PROGRAM Fixt2_Seq_Call
VAR
	Clamp_1: FB_CylinderModule;
	Clamp_2: FB_CylinderModule;
	Clamp_3: FB_CylinderModule;
	Clamp_4: FB_CylinderModule;
	Clamp_5: FB_CylinderModule;
	Clamp_6: FB_CylinderModule;
	sAlwaysoff: BOOL;
	FB_AutoSeq_0: FB_AutoSeq;
	alwayson:BOOL;
	partmonitor:FB_PartMonitoring_fixt2;
	trunion:FB_Trunion;
END_VAR
VAR // added by the converter: edge detectors and wires of the graphical bodies
    _w1, _w2, _w3, _w4, _w5, _w6 : BOOL;
END_VAR

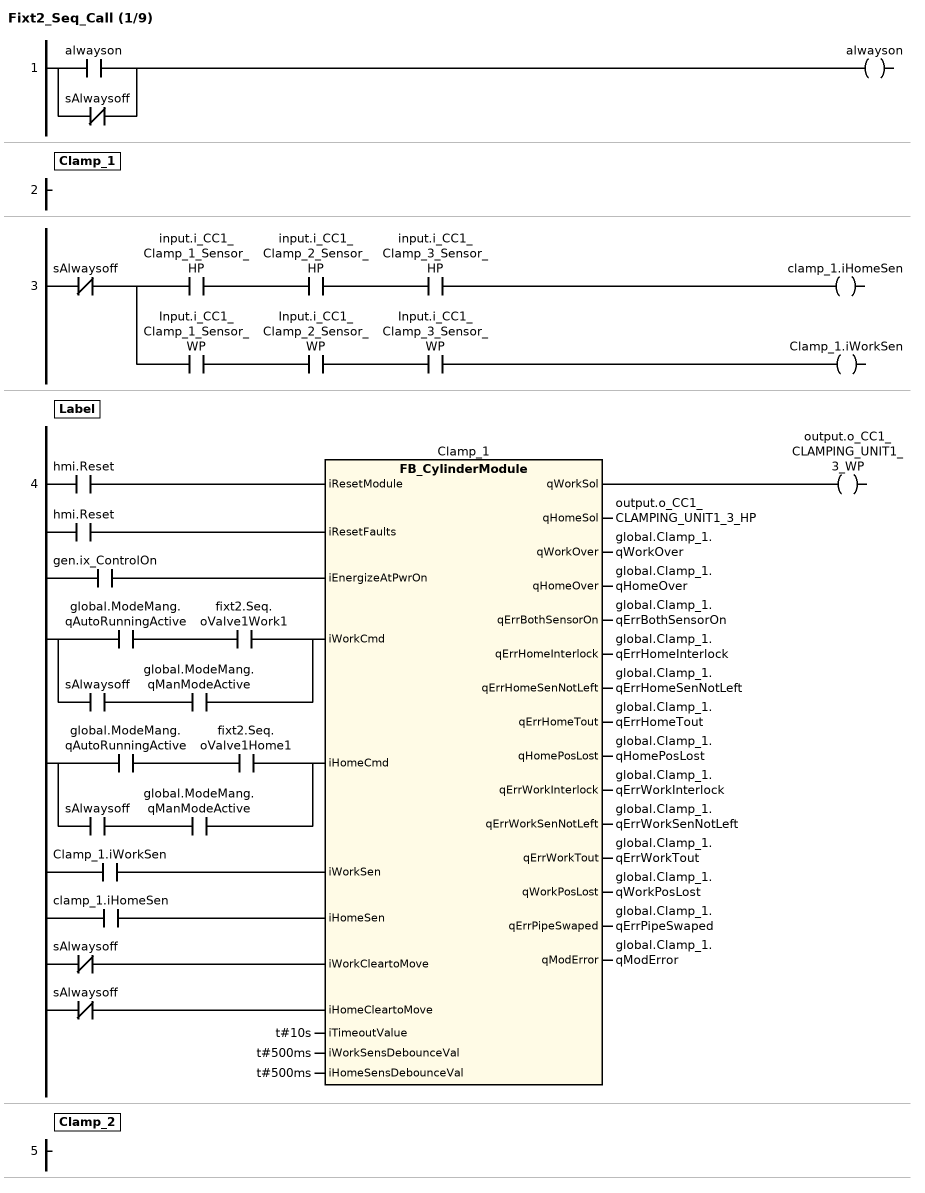
// NETWORK 1
alwayson := alwayson OR NOT sAlwaysoff;

// NETWORK 2
Clamp_1: ;

// NETWORK 3
_w1 := NOT sAlwaysoff;
clamp_1.iHomeSen := _w1 AND input.i_CC1_Clamp_1_Sensor_HP AND input.i_CC1_Clamp_2_Sensor_HP AND input.i_CC1_Clamp_3_Sensor_HP;
Clamp_1.iWorkSen := _w1 AND Input.i_CC1_Clamp_1_Sensor_WP AND Input.i_CC1_Clamp_2_Sensor_WP AND Input.i_CC1_Clamp_3_Sensor_WP;

// NETWORK 4
Label:
Clamp_1(
    iResetModule := hmi.Reset,
    iResetFaults := hmi.Reset,
    iEnergizeAtPwrOn := gen.ix_ControlOn,
    iWorkCmd := global.ModeMang.qAutoRunningActive AND fixt2.Seq.oValve1Work1 OR sAlwaysoff AND global.ModeMang.qManModeActive,
    iHomeCmd := global.ModeMang.qAutoRunningActive AND fixt2.Seq.oValve1Home1 OR sAlwaysoff AND global.ModeMang.qManModeActive,
    iWorkSen := Clamp_1.iWorkSen,
    iHomeSen := clamp_1.iHomeSen,
    iWorkCleartoMove := NOT sAlwaysoff,
    iHomeCleartoMove := NOT sAlwaysoff,
    iTimeoutValue := t#10s,
    iWorkSensDebounceVal := t#500ms,
    iHomeSensDebounceVal := t#500ms,
    qHomeSol => output.o_CC1_CLAMPING_UNIT1_3_HP,
    qWorkOver => global.Clamp_1.qWorkOver,
    qHomeOver => global.Clamp_1.qHomeOver,
    qErrBothSensorOn => global.Clamp_1.qErrBothSensorOn,
    qErrHomeInterlock => global.Clamp_1.qErrHomeInterlock,
    qErrHomeSenNotLeft => global.Clamp_1.qErrHomeSenNotLeft,
    qErrHomeTout => global.Clamp_1.qErrHomeTout,
    qHomePosLost => global.Clamp_1.qHomePosLost,
    qErrWorkInterlock => global.Clamp_1.qErrWorkInterlock,
    qErrWorkSenNotLeft => global.Clamp_1.qErrWorkSenNotLeft,
    qErrWorkTout => global.Clamp_1.qErrWorkTout,
    qWorkPosLost => global.Clamp_1.qWorkPosLost,
    qErrPipeSwaped => global.Clamp_1.qErrPipeSwaped,
    qModError => global.Clamp_1.qModError); // FB_CylinderModule
output.o_CC1_CLAMPING_UNIT1_3_WP := Clamp_1.qWorkSol;

// NETWORK 5
Clamp_2: ;

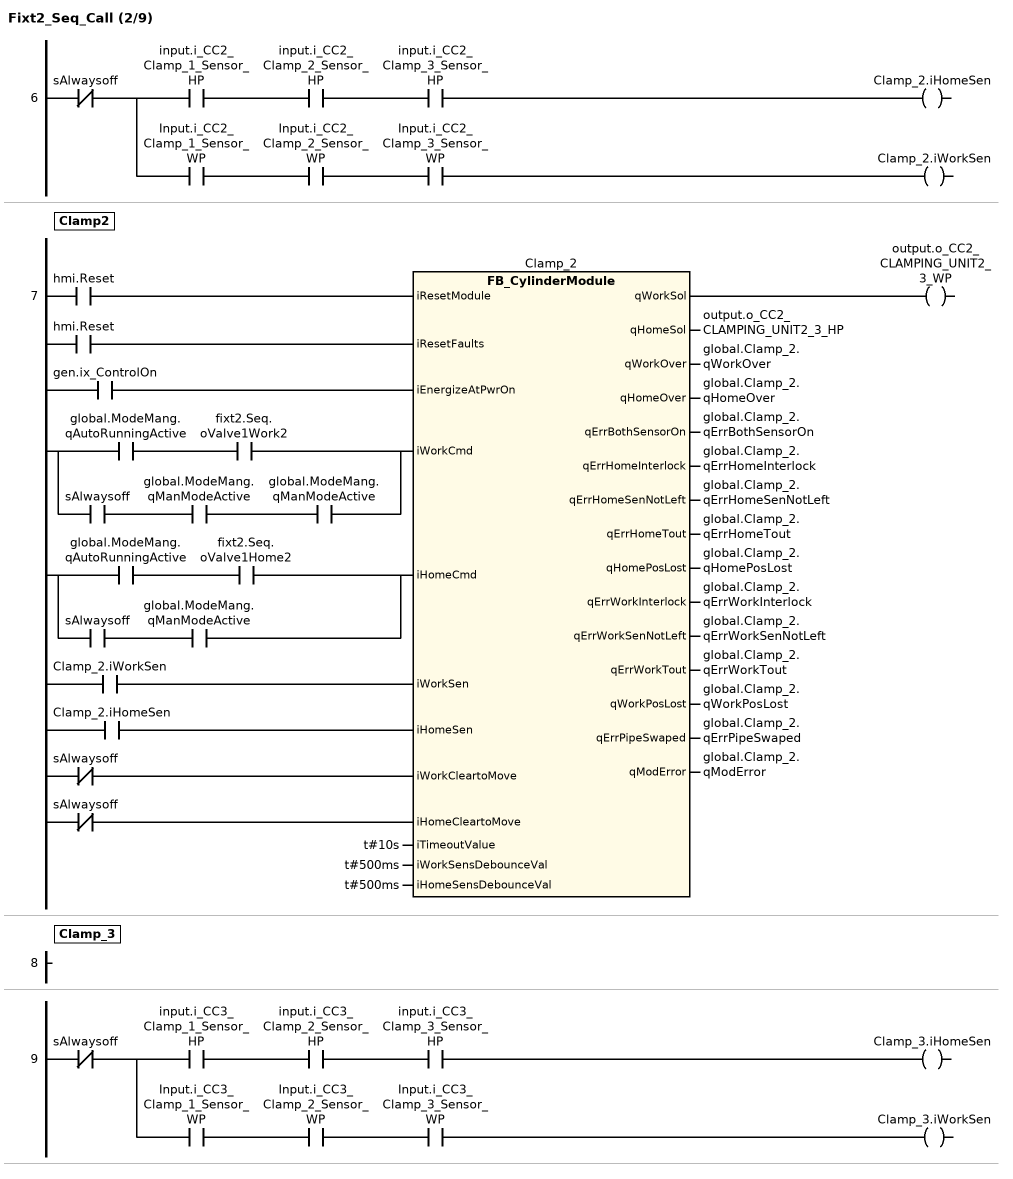
// NETWORK 6
_w2 := NOT sAlwaysoff;
Clamp_2.iHomeSen := _w2 AND input.i_CC2_Clamp_1_Sensor_HP AND input.i_CC2_Clamp_2_Sensor_HP AND input.i_CC2_Clamp_3_Sensor_HP;
Clamp_2.iWorkSen := _w2 AND Input.i_CC2_Clamp_1_Sensor_WP AND Input.i_CC2_Clamp_2_Sensor_WP AND Input.i_CC2_Clamp_3_Sensor_WP;

// NETWORK 7
Clamp2:
Clamp_2(
    iResetModule := hmi.Reset,
    iResetFaults := hmi.Reset,
    iEnergizeAtPwrOn := gen.ix_ControlOn,
    iWorkCmd := global.ModeMang.qAutoRunningActive AND fixt2.Seq.oValve1Work2 OR sAlwaysoff AND global.ModeMang.qManModeActive AND global.ModeMang.qManModeActive,
    iHomeCmd := global.ModeMang.qAutoRunningActive AND fixt2.Seq.oValve1Home2 OR sAlwaysoff AND global.ModeMang.qManModeActive,
    iWorkSen := Clamp_2.iWorkSen,
    iHomeSen := Clamp_2.iHomeSen,
    iWorkCleartoMove := NOT sAlwaysoff,
    iHomeCleartoMove := NOT sAlwaysoff,
    iTimeoutValue := t#10s,
    iWorkSensDebounceVal := t#500ms,
    iHomeSensDebounceVal := t#500ms,
    qHomeSol => output.o_CC2_CLAMPING_UNIT2_3_HP,
    qWorkOver => global.Clamp_2.qWorkOver,
    qHomeOver => global.Clamp_2.qHomeOver,
    qErrBothSensorOn => global.Clamp_2.qErrBothSensorOn,
    qErrHomeInterlock => global.Clamp_2.qErrHomeInterlock,
    qErrHomeSenNotLeft => global.Clamp_2.qErrHomeSenNotLeft,
    qErrHomeTout => global.Clamp_2.qErrHomeTout,
    qHomePosLost => global.Clamp_2.qHomePosLost,
    qErrWorkInterlock => global.Clamp_2.qErrWorkInterlock,
    qErrWorkSenNotLeft => global.Clamp_2.qErrWorkSenNotLeft,
    qErrWorkTout => global.Clamp_2.qErrWorkTout,
    qWorkPosLost => global.Clamp_2.qWorkPosLost,
    qErrPipeSwaped => global.Clamp_2.qErrPipeSwaped,
    qModError => global.Clamp_2.qModError); // FB_CylinderModule
output.o_CC2_CLAMPING_UNIT2_3_WP := Clamp_2.qWorkSol;

// NETWORK 8
Clamp_3: ;

// NETWORK 9
_w3 := NOT sAlwaysoff;
Clamp_3.iHomeSen := _w3 AND input.i_CC3_Clamp_1_Sensor_HP AND input.i_CC3_Clamp_2_Sensor_HP AND input.i_CC3_Clamp_3_Sensor_HP;
Clamp_3.iWorkSen := _w3 AND Input.i_CC3_Clamp_1_Sensor_WP AND Input.i_CC3_Clamp_2_Sensor_WP AND Input.i_CC3_Clamp_3_Sensor_WP;

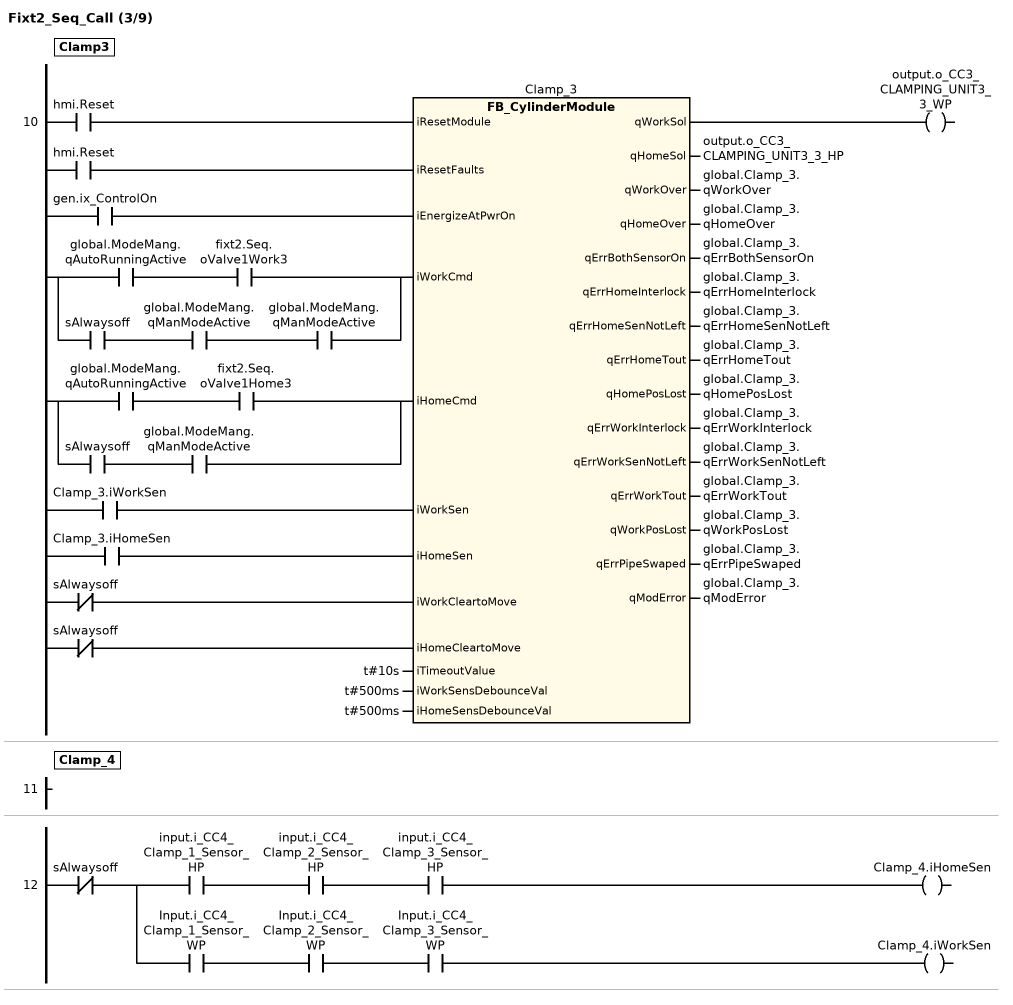
// NETWORK 10
Clamp3:
Clamp_3(
    iResetModule := hmi.Reset,
    iResetFaults := hmi.Reset,
    iEnergizeAtPwrOn := gen.ix_ControlOn,
    iWorkCmd := global.ModeMang.qAutoRunningActive AND fixt2.Seq.oValve1Work3 OR sAlwaysoff AND global.ModeMang.qManModeActive AND global.ModeMang.qManModeActive,
    iHomeCmd := global.ModeMang.qAutoRunningActive AND fixt2.Seq.oValve1Home3 OR sAlwaysoff AND global.ModeMang.qManModeActive,
    iWorkSen := Clamp_3.iWorkSen,
    iHomeSen := Clamp_3.iHomeSen,
    iWorkCleartoMove := NOT sAlwaysoff,
    iHomeCleartoMove := NOT sAlwaysoff,
    iTimeoutValue := t#10s,
    iWorkSensDebounceVal := t#500ms,
    iHomeSensDebounceVal := t#500ms,
    qHomeSol => output.o_CC3_CLAMPING_UNIT3_3_HP,
    qWorkOver => global.Clamp_3.qWorkOver,
    qHomeOver => global.Clamp_3.qHomeOver,
    qErrBothSensorOn => global.Clamp_3.qErrBothSensorOn,
    qErrHomeInterlock => global.Clamp_3.qErrHomeInterlock,
    qErrHomeSenNotLeft => global.Clamp_3.qErrHomeSenNotLeft,
    qErrHomeTout => global.Clamp_3.qErrHomeTout,
    qHomePosLost => global.Clamp_3.qHomePosLost,
    qErrWorkInterlock => global.Clamp_3.qErrWorkInterlock,
    qErrWorkSenNotLeft => global.Clamp_3.qErrWorkSenNotLeft,
    qErrWorkTout => global.Clamp_3.qErrWorkTout,
    qWorkPosLost => global.Clamp_3.qWorkPosLost,
    qErrPipeSwaped => global.Clamp_3.qErrPipeSwaped,
    qModError => global.Clamp_3.qModError); // FB_CylinderModule
output.o_CC3_CLAMPING_UNIT3_3_WP := Clamp_3.qWorkSol;

// NETWORK 11
Clamp_4: ;

// NETWORK 12
_w4 := NOT sAlwaysoff;
Clamp_4.iHomeSen := _w4 AND input.i_CC4_Clamp_1_Sensor_HP AND input.i_CC4_Clamp_2_Sensor_HP AND input.i_CC4_Clamp_3_Sensor_HP;
Clamp_4.iWorkSen := _w4 AND Input.i_CC4_Clamp_1_Sensor_WP AND Input.i_CC4_Clamp_2_Sensor_WP AND Input.i_CC4_Clamp_3_Sensor_WP;

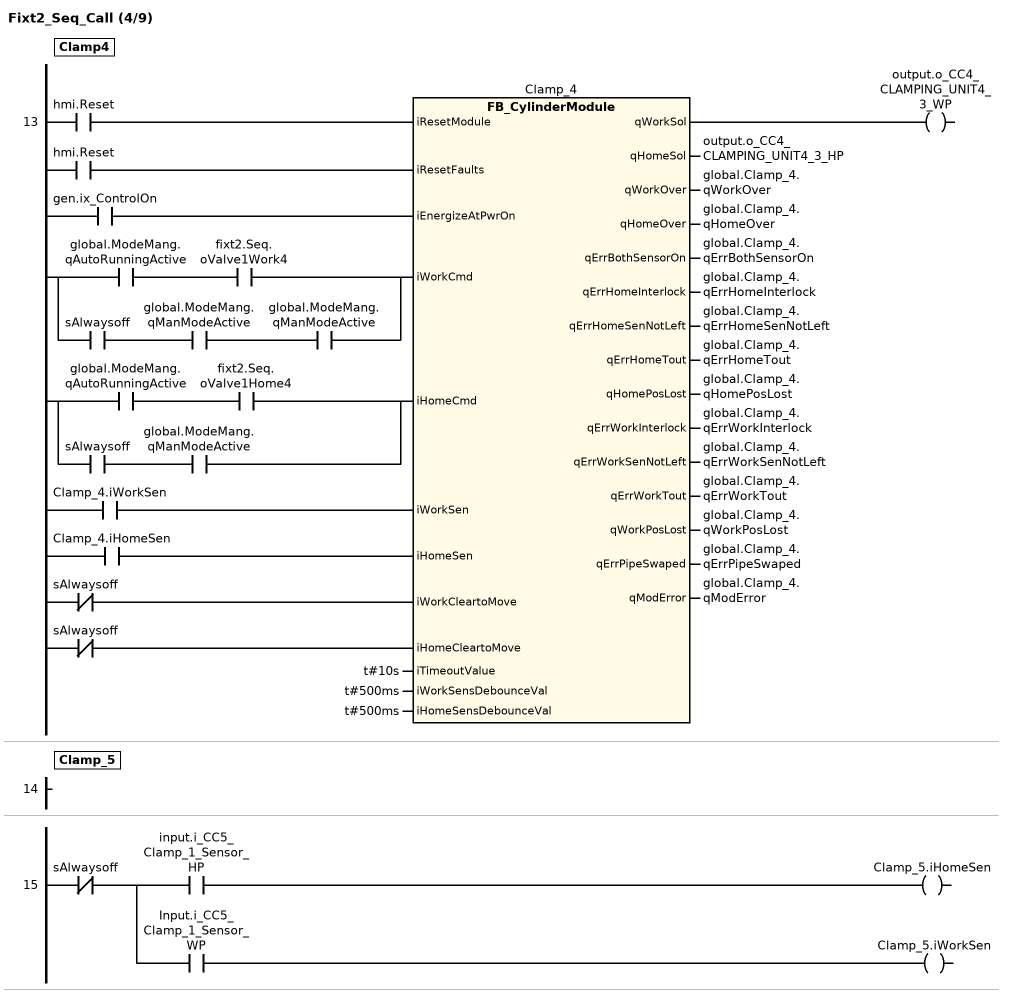
// NETWORK 13
Clamp4:
Clamp_4(
    iResetModule := hmi.Reset,
    iResetFaults := hmi.Reset,
    iEnergizeAtPwrOn := gen.ix_ControlOn,
    iWorkCmd := global.ModeMang.qAutoRunningActive AND fixt2.Seq.oValve1Work4 OR sAlwaysoff AND global.ModeMang.qManModeActive AND global.ModeMang.qManModeActive,
    iHomeCmd := global.ModeMang.qAutoRunningActive AND fixt2.Seq.oValve1Home4 OR sAlwaysoff AND global.ModeMang.qManModeActive,
    iWorkSen := Clamp_4.iWorkSen,
    iHomeSen := Clamp_4.iHomeSen,
    iWorkCleartoMove := NOT sAlwaysoff,
    iHomeCleartoMove := NOT sAlwaysoff,
    iTimeoutValue := t#10s,
    iWorkSensDebounceVal := t#500ms,
    iHomeSensDebounceVal := t#500ms,
    qHomeSol => output.o_CC4_CLAMPING_UNIT4_3_HP,
    qWorkOver => global.Clamp_4.qWorkOver,
    qHomeOver => global.Clamp_4.qHomeOver,
    qErrBothSensorOn => global.Clamp_4.qErrBothSensorOn,
    qErrHomeInterlock => global.Clamp_4.qErrHomeInterlock,
    qErrHomeSenNotLeft => global.Clamp_4.qErrHomeSenNotLeft,
    qErrHomeTout => global.Clamp_4.qErrHomeTout,
    qHomePosLost => global.Clamp_4.qHomePosLost,
    qErrWorkInterlock => global.Clamp_4.qErrWorkInterlock,
    qErrWorkSenNotLeft => global.Clamp_4.qErrWorkSenNotLeft,
    qErrWorkTout => global.Clamp_4.qErrWorkTout,
    qWorkPosLost => global.Clamp_4.qWorkPosLost,
    qErrPipeSwaped => global.Clamp_4.qErrPipeSwaped,
    qModError => global.Clamp_4.qModError); // FB_CylinderModule
output.o_CC4_CLAMPING_UNIT4_3_WP := Clamp_4.qWorkSol;

// NETWORK 14
Clamp_5: ;

// NETWORK 15
_w5 := NOT sAlwaysoff;
Clamp_5.iHomeSen := _w5 AND input.i_CC5_Clamp_1_Sensor_HP;
Clamp_5.iWorkSen := _w5 AND Input.i_CC5_Clamp_1_Sensor_WP;

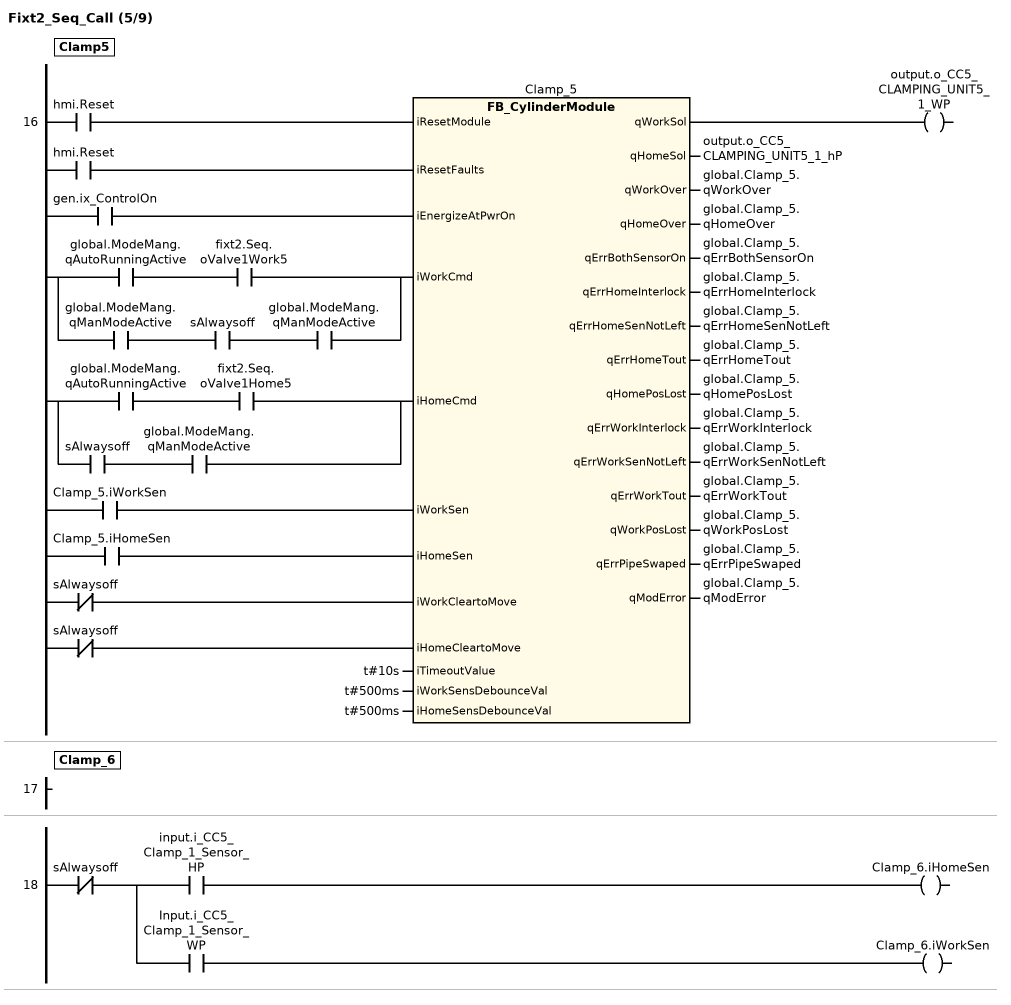
// NETWORK 16
Clamp5:
Clamp_5(
    iResetModule := hmi.Reset,
    iResetFaults := hmi.Reset,
    iEnergizeAtPwrOn := gen.ix_ControlOn,
    iWorkCmd := global.ModeMang.qAutoRunningActive AND fixt2.Seq.oValve1Work5 OR global.ModeMang.qManModeActive AND sAlwaysoff AND global.ModeMang.qManModeActive,
    iHomeCmd := global.ModeMang.qAutoRunningActive AND fixt2.Seq.oValve1Home5 OR sAlwaysoff AND global.ModeMang.qManModeActive,
    iWorkSen := Clamp_5.iWorkSen,
    iHomeSen := Clamp_5.iHomeSen,
    iWorkCleartoMove := NOT sAlwaysoff,
    iHomeCleartoMove := NOT sAlwaysoff,
    iTimeoutValue := t#10s,
    iWorkSensDebounceVal := t#500ms,
    iHomeSensDebounceVal := t#500ms,
    qHomeSol => output.o_CC5_CLAMPING_UNIT5_1_hP,
    qWorkOver => global.Clamp_5.qWorkOver,
    qHomeOver => global.Clamp_5.qHomeOver,
    qErrBothSensorOn => global.Clamp_5.qErrBothSensorOn,
    qErrHomeInterlock => global.Clamp_5.qErrHomeInterlock,
    qErrHomeSenNotLeft => global.Clamp_5.qErrHomeSenNotLeft,
    qErrHomeTout => global.Clamp_5.qErrHomeTout,
    qHomePosLost => global.Clamp_5.qHomePosLost,
    qErrWorkInterlock => global.Clamp_5.qErrWorkInterlock,
    qErrWorkSenNotLeft => global.Clamp_5.qErrWorkSenNotLeft,
    qErrWorkTout => global.Clamp_5.qErrWorkTout,
    qWorkPosLost => global.Clamp_5.qWorkPosLost,
    qErrPipeSwaped => global.Clamp_5.qErrPipeSwaped,
    qModError => global.Clamp_5.qModError); // FB_CylinderModule
output.o_CC5_CLAMPING_UNIT5_1_WP := Clamp_5.qWorkSol;

// NETWORK 17
Clamp_6: ;

// NETWORK 18
_w6 := NOT sAlwaysoff;
Clamp_6.iHomeSen := _w6 AND input.i_CC5_Clamp_1_Sensor_HP;
Clamp_6.iWorkSen := _w6 AND Input.i_CC5_Clamp_1_Sensor_WP;

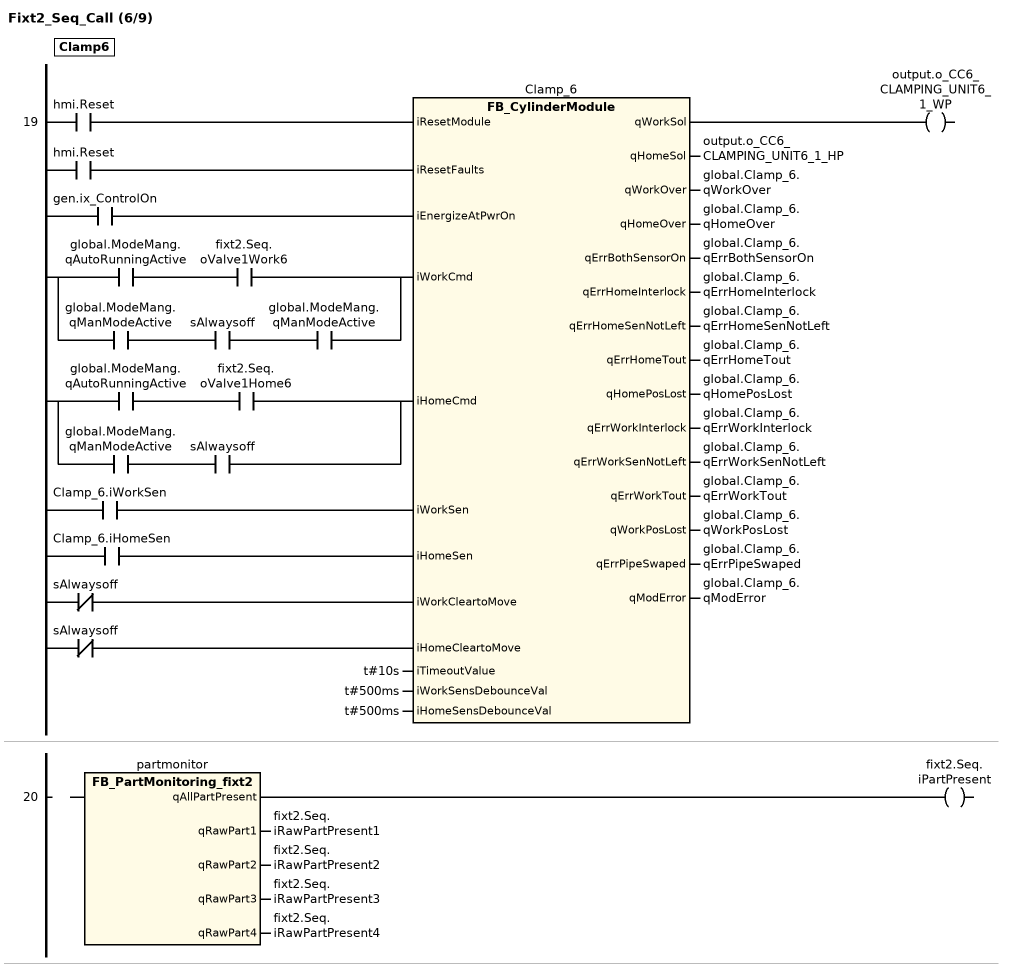
// NETWORK 19
Clamp6:
Clamp_6(
    iResetModule := hmi.Reset,
    iResetFaults := hmi.Reset,
    iEnergizeAtPwrOn := gen.ix_ControlOn,
    iWorkCmd := global.ModeMang.qAutoRunningActive AND fixt2.Seq.oValve1Work6 OR global.ModeMang.qManModeActive AND sAlwaysoff AND global.ModeMang.qManModeActive,
    iHomeCmd := global.ModeMang.qAutoRunningActive AND fixt2.Seq.oValve1Home6 OR global.ModeMang.qManModeActive AND sAlwaysoff,
    iWorkSen := Clamp_6.iWorkSen,
    iHomeSen := Clamp_6.iHomeSen,
    iWorkCleartoMove := NOT sAlwaysoff,
    iHomeCleartoMove := NOT sAlwaysoff,
    iTimeoutValue := t#10s,
    iWorkSensDebounceVal := t#500ms,
    iHomeSensDebounceVal := t#500ms,
    qHomeSol => output.o_CC6_CLAMPING_UNIT6_1_HP,
    qWorkOver => global.Clamp_6.qWorkOver,
    qHomeOver => global.Clamp_6.qHomeOver,
    qErrBothSensorOn => global.Clamp_6.qErrBothSensorOn,
    qErrHomeInterlock => global.Clamp_6.qErrHomeInterlock,
    qErrHomeSenNotLeft => global.Clamp_6.qErrHomeSenNotLeft,
    qErrHomeTout => global.Clamp_6.qErrHomeTout,
    qHomePosLost => global.Clamp_6.qHomePosLost,
    qErrWorkInterlock => global.Clamp_6.qErrWorkInterlock,
    qErrWorkSenNotLeft => global.Clamp_6.qErrWorkSenNotLeft,
    qErrWorkTout => global.Clamp_6.qErrWorkTout,
    qWorkPosLost => global.Clamp_6.qWorkPosLost,
    qErrPipeSwaped => global.Clamp_6.qErrPipeSwaped,
    qModError => global.Clamp_6.qModError); // FB_CylinderModule
output.o_CC6_CLAMPING_UNIT6_1_WP := Clamp_6.qWorkSol;

// NETWORK 20
partmonitor(
    qRawPart1 => fixt2.Seq.iRawPartPresent1,
    qRawPart2 => fixt2.Seq.iRawPartPresent2,
    qRawPart3 => fixt2.Seq.iRawPartPresent3,
    qRawPart4 => fixt2.Seq.iRawPartPresent4); // FB_PartMonitoring_fixt2
fixt2.Seq.iPartPresent := partmonitor.qAllPartPresent;

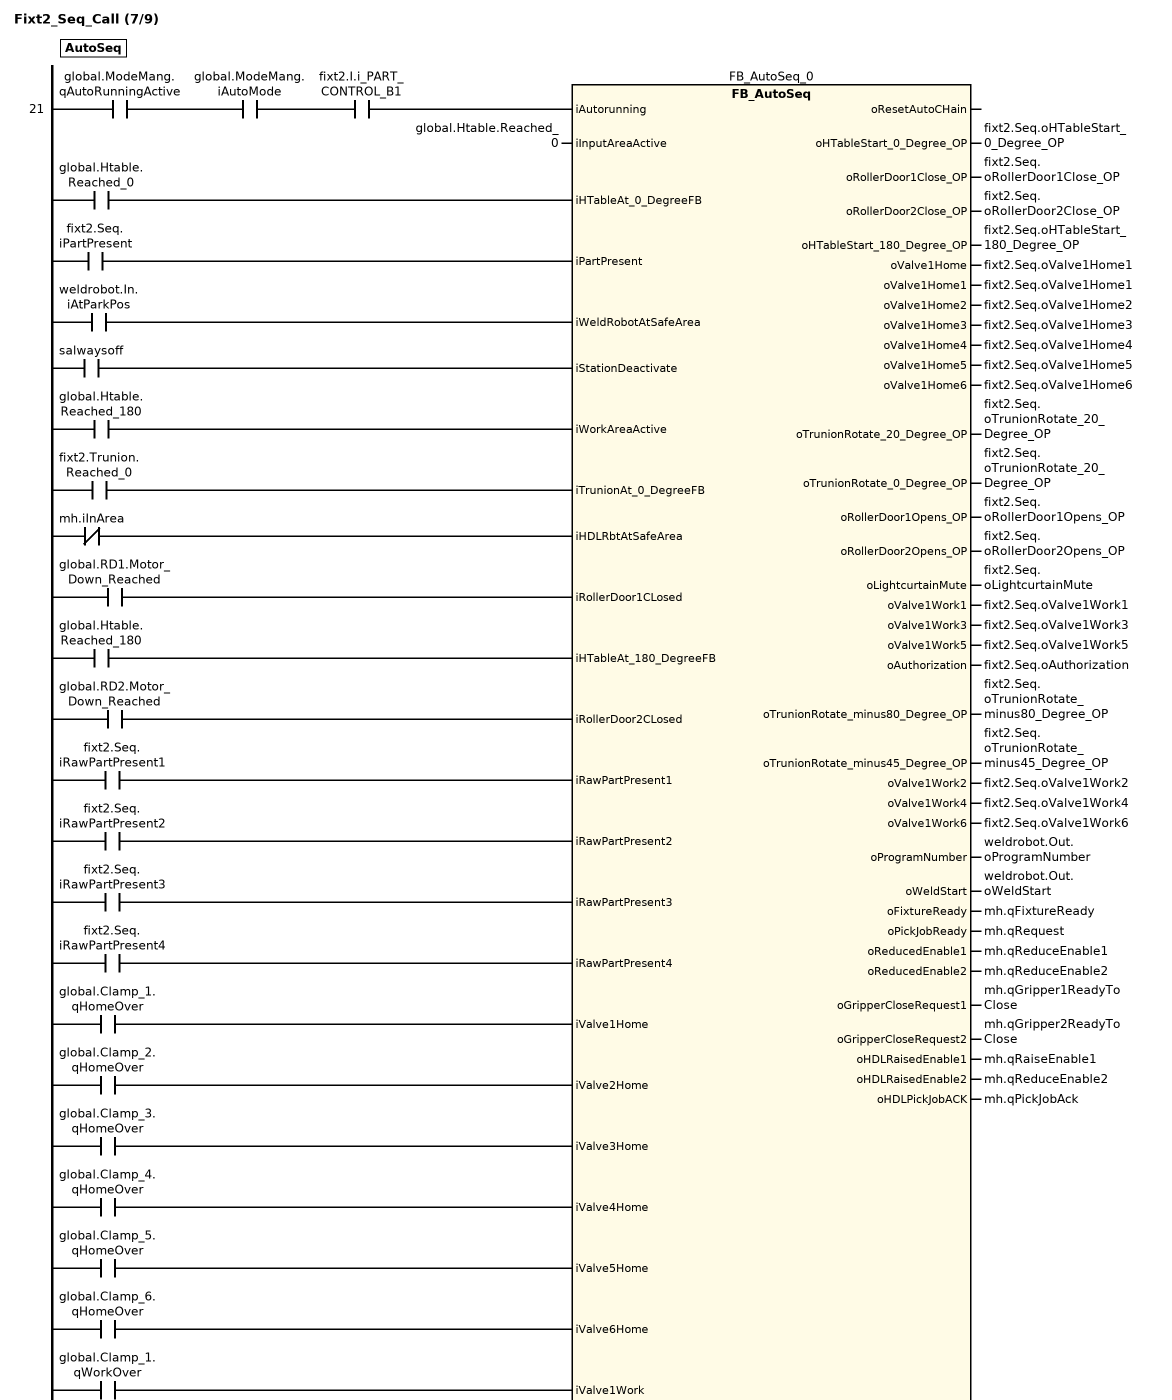
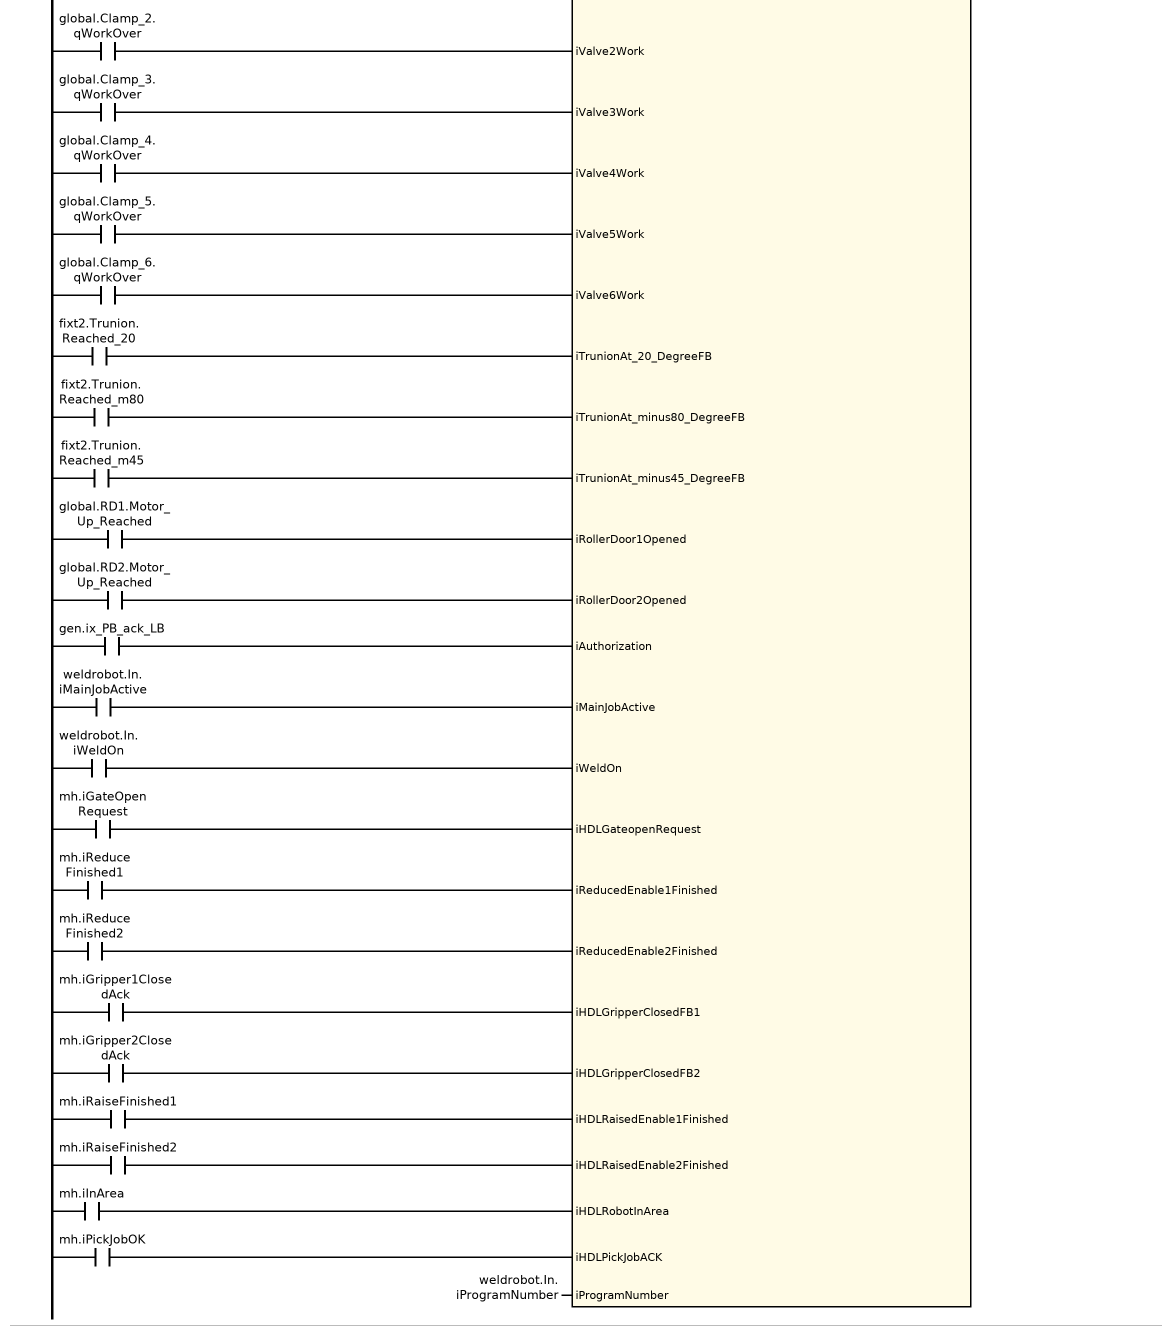
// NETWORK 21
AutoSeq:
FB_AutoSeq_0(
    iAutorunning := global.ModeMang.qAutoRunningActive AND global.ModeMang.iAutoMode AND fixt2.I.i_PART_CONTROL_B1,
    iInputAreaActive := global.Htable.Reached_0,
    iHTableAt_0_DegreeFB := global.Htable.Reached_0,
    iPartPresent := fixt2.Seq.iPartPresent,
    iWeldRobotAtSafeArea := weldrobot.In.iAtParkPos,
    iStationDeactivate := salwaysoff,
    iWorkAreaActive := global.Htable.Reached_180,
    iTrunionAt_0_DegreeFB := fixt2.Trunion.Reached_0,
    iHDLRbtAtSafeArea := NOT mh.iInArea,
    iRollerDoor1CLosed := global.RD1.Motor_Down_Reached,
    iHTableAt_180_DegreeFB := global.Htable.Reached_180,
    iRollerDoor2CLosed := global.RD2.Motor_Down_Reached,
    iRawPartPresent1 := fixt2.Seq.iRawPartPresent1,
    iRawPartPresent2 := fixt2.Seq.iRawPartPresent2,
    iRawPartPresent3 := fixt2.Seq.iRawPartPresent3,
    iRawPartPresent4 := fixt2.Seq.iRawPartPresent4,
    iValve1Home := global.Clamp_1.qHomeOver,
    iValve2Home := global.Clamp_2.qHomeOver,
    iValve3Home := global.Clamp_3.qHomeOver,
    iValve4Home := global.Clamp_4.qHomeOver,
    iValve5Home := global.Clamp_5.qHomeOver,
    iValve6Home := global.Clamp_6.qHomeOver,
    iValve1Work := global.Clamp_1.qWorkOver,
    iValve2Work := global.Clamp_2.qWorkOver,
    iValve3Work := global.Clamp_3.qWorkOver,
    iValve4Work := global.Clamp_4.qWorkOver,
    iValve5Work := global.Clamp_5.qWorkOver,
    iValve6Work := global.Clamp_6.qWorkOver,
    iTrunionAt_20_DegreeFB := fixt2.Trunion.Reached_20,
    iTrunionAt_minus80_DegreeFB := fixt2.Trunion.Reached_m80,
    iTrunionAt_minus45_DegreeFB := fixt2.Trunion.Reached_m45,
    iRollerDoor1Opened := global.RD1.Motor_Up_Reached,
    iRollerDoor2Opened := global.RD2.Motor_Up_Reached,
    iAuthorization := gen.ix_PB_ack_LB,
    iMainJobActive := weldrobot.In.iMainJobActive,
    iWeldOn := weldrobot.In.iWeldOn,
    iHDLGateopenRequest := mh.iGateOpenRequest,
    iReducedEnable1Finished := mh.iReduceFinished1,
    iReducedEnable2Finished := mh.iReduceFinished2,
    iHDLGripperClosedFB1 := mh.iGripper1ClosedAck,
    iHDLGripperClosedFB2 := mh.iGripper2ClosedAck,
    iHDLRaisedEnable1Finished := mh.iRaiseFinished1,
    iHDLRaisedEnable2Finished := mh.iRaiseFinished2,
    iHDLRobotInArea := mh.iInArea,
    iHDLPickJobACK := mh.iPickJobOK,
    iProgramNumber := weldrobot.In.iProgramNumber,
    oHTableStart_0_Degree_OP => fixt2.Seq.oHTableStart_0_Degree_OP,
    oRollerDoor1Close_OP => fixt2.Seq.oRollerDoor1Close_OP,
    oRollerDoor2Close_OP => fixt2.Seq.oRollerDoor2Close_OP,
    oHTableStart_180_Degree_OP => fixt2.Seq.oHTableStart_180_Degree_OP,
    oValve1Home => fixt2.Seq.oValve1Home1,
    oValve1Home1 => fixt2.Seq.oValve1Home1,
    oValve1Home2 => fixt2.Seq.oValve1Home2,
    oValve1Home3 => fixt2.Seq.oValve1Home3,
    oValve1Home4 => fixt2.Seq.oValve1Home4,
    oValve1Home5 => fixt2.Seq.oValve1Home5,
    oValve1Home6 => fixt2.Seq.oValve1Home6,
    oTrunionRotate_20_Degree_OP => fixt2.Seq.oTrunionRotate_20_Degree_OP,
    oTrunionRotate_0_Degree_OP => fixt2.Seq.oTrunionRotate_20_Degree_OP,
    oRollerDoor1Opens_OP => fixt2.Seq.oRollerDoor1Opens_OP,
    oRollerDoor2Opens_OP => fixt2.Seq.oRollerDoor2Opens_OP,
    oLightcurtainMute => fixt2.Seq.oLightcurtainMute,
    oValve1Work1 => fixt2.Seq.oValve1Work1,
    oValve1Work3 => fixt2.Seq.oValve1Work3,
    oValve1Work5 => fixt2.Seq.oValve1Work5,
    oAuthorization => fixt2.Seq.oAuthorization,
    oTrunionRotate_minus80_Degree_OP => fixt2.Seq.oTrunionRotate_minus80_Degree_OP,
    oTrunionRotate_minus45_Degree_OP => fixt2.Seq.oTrunionRotate_minus45_Degree_OP,
    oValve1Work2 => fixt2.Seq.oValve1Work2,
    oValve1Work4 => fixt2.Seq.oValve1Work4,
    oValve1Work6 => fixt2.Seq.oValve1Work6,
    oProgramNumber => weldrobot.Out.oProgramNumber,
    oWeldStart => weldrobot.Out.oWeldStart,
    oFixtureReady => mh.qFixtureReady,
    oPickJobReady => mh.qRequest,
    oReducedEnable1 => mh.qReduceEnable1,
    oReducedEnable2 => mh.qReduceEnable2,
    oGripperCloseRequest1 => mh.qGripper1ReadyToClose,
    oGripperCloseRequest2 => mh.qGripper2ReadyToClose,
    oHDLRaisedEnable1 => mh.qRaiseEnable1,
    oHDLRaisedEnable2 => mh.qReduceEnable2,
    oHDLPickJobACK => mh.qPickJobAck); // FB_AutoSeq

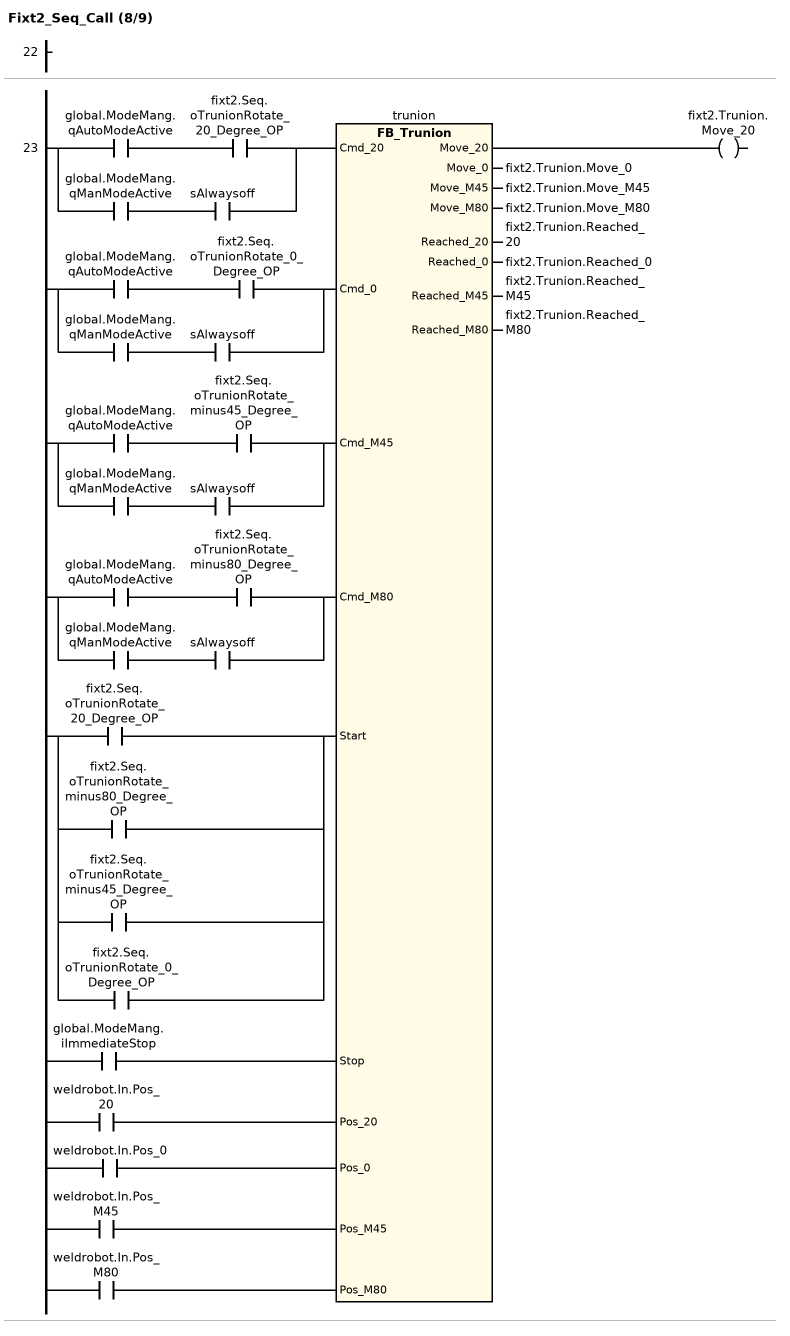
// NETWORK 22

// NETWORK 23
trunion(
    Cmd_20 := global.ModeMang.qAutoModeActive AND fixt2.Seq.oTrunionRotate_20_Degree_OP OR global.ModeMang.qManModeActive AND sAlwaysoff,
    Cmd_0 := global.ModeMang.qAutoModeActive AND fixt2.Seq.oTrunionRotate_0_Degree_OP OR global.ModeMang.qManModeActive AND sAlwaysoff,
    Cmd_M45 := global.ModeMang.qAutoModeActive AND fixt2.Seq.oTrunionRotate_minus45_Degree_OP OR global.ModeMang.qManModeActive AND sAlwaysoff,
    Cmd_M80 := global.ModeMang.qAutoModeActive AND fixt2.Seq.oTrunionRotate_minus80_Degree_OP OR global.ModeMang.qManModeActive AND sAlwaysoff,
    Start := fixt2.Seq.oTrunionRotate_20_Degree_OP OR fixt2.Seq.oTrunionRotate_minus80_Degree_OP OR fixt2.Seq.oTrunionRotate_minus45_Degree_OP OR fixt2.Seq.oTrunionRotate_0_Degree_OP,
    Stop := global.ModeMang.iImmediateStop,
    Pos_20 := weldrobot.In.Pos_20,
    Pos_0 := weldrobot.In.Pos_0,
    Pos_M45 := weldrobot.In.Pos_M45,
    Pos_M80 := weldrobot.In.Pos_M80,
    Move_0 => fixt2.Trunion.Move_0,
    Move_M45 => fixt2.Trunion.Move_M45,
    Move_M80 => fixt2.Trunion.Move_M80,
    Reached_20 => fixt2.Trunion.Reached_20,
    Reached_0 => fixt2.Trunion.Reached_0,
    Reached_M45 => fixt2.Trunion.Reached_M45,
    Reached_M80 => fixt2.Trunion.Reached_M80); // FB_Trunion
fixt2.Trunion.Move_20 := trunion.Move_20;

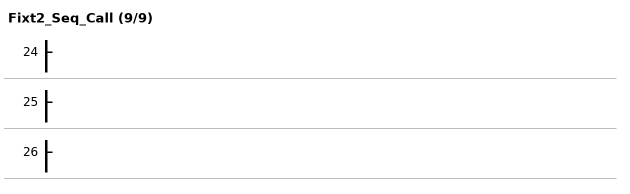
// NETWORK 24

// NETWORK 25

// NETWORK 26

END_PROGRAM

(* stored: Version 1.1.0.1, ProductVersion 3.1.4024.16
   POU Fixt2_Seq_Call: Id {5ad8aca1-aa2e-4469-8e83-babea9984baf}, SpecialFunc None *)
